INTERFACE I_LogBuilder

METHOD CreateLog
END_METHOD

METHOD WithContextInt : I_LogBuilder
VAR_INPUT
	sName		: T_MaxString;
	nValue		: INT;
END_VAR
END_METHOD

METHOD WithIntArg : I_LogBuilder
VAR_INPUT
	nValue		: INT;
END_VAR
END_METHOD

METHOD WithLogger : I_LogBuilder
VAR_INPUT
	sLogger		: T_MaxString;
END_VAR
END_METHOD

METHOD WithStringArg : I_LogBuilder
VAR_INPUT
	sValue		: T_MaxString;
END_VAR
END_METHOD

END_INTERFACE

(* stored: Version 1.1.0.1, ProductVersion 3.1.4024.0
   Itf I_LogBuilder: Id {7cc70285-5d0d-45bd-9ca5-5fc75d169d66}
   Method CreateLog: Id {d4566474-f2a6-454e-aec0-dcc53c0a7142}
   Method WithContextInt: Id {afc2f3dd-7c7d-4dac-b12b-9815415ba0cf}
   Method WithIntArg: Id {f92f2c8f-a7cf-4fc5-88d4-0a0f0c6c46ad}
   Method WithLogger: Id {16cc3ca7-f012-48b3-9f1b-77ccafb03fbc}
   Method WithStringArg: Id {8e3c58b9-db8c-4af2-b60b-bf29d4e372e6} *)
